Staubli VAL3: range.pgx

public program range(num x_nStart, num x_nEnd, num x_nStep, num& x_nResult[])
  local num l_nCoutner
  local num l_nElement
begin

  l_nCoutner = 0
  resize(x_nResult,1,1)
  x_nResult = 0

  for l_nElement = x_nStart to x_nEnd-1 step x_nStep
    l_nCoutner = l_nCoutner+1
    append(x_nResult)
    x_nResult[l_nCoutner] = l_nElement
  endFor

  delete(x_nResult[0])

end
